(* CODESYS project IoDrvSubModulesSlotTest.project

Project tree, tasks and I/O mapping:
  Device : CODESYS Control Win V3, 3S - Smart Software Solutions GmbH, order no. 305021, version 3.5.9.0
    application Application
      libraries: Standard, * (System)
      task MainTask (cyclic, interval t#20ms, priority 1) calls PLC_PRG
      program PLC_PRG [ST]
    IoDrvSubModulesSlot : IoDrvSubModulesSlot, MyCompany, order no. 4711, version 3.5.9.0
      SubModuleForSlotConnector : SubModuleForSlotConnector, MyCompany, order no. abc, version 3.5.9.0
          output out1 : BYTE  // out1
          unmapped channels: out2
      SlotSubModuleAsLocalModule : SlotSubModuleAsLocalModule, MyCompany, order no. abc, version 3.5.9.0
          input  in1 : BYTE  // in1
          unmapped channels: in2
      <Empty>
      <Empty>
      <Empty>
      <Empty>
      <Empty>
      <Empty>
*)

// Device/Application/PLC_PRG
PROGRAM PLC_PRG
VAR
END_VAR

(* Let the output run. *)
out1 := out1 + 1;
(* input us updated by IO driver *)
in1;

END_PROGRAM
